(* IEC 61131-3 sources: Eaton-PLC-CSV-MQTT/CSV-MQTT/scripts/FunctionBlocks, 2 files *)

(* ---- FB_CSVReader.st ---- *)
// This function block reads CSV files row by row for PLC processing
// Uses state machine approach for efficient file handling
FUNCTION_BLOCK FB_CSVReader
VAR_INPUT
    xEnable   : BOOL;   // TRUE = start/continue reading, FALSE = stop and reset
    sFilePath : STRING; // File path to the CSV file (e.g., '/usr/data.csv')
END_VAR
VAR_OUTPUT
    RowOut    : ST_CSVRow; // Output: One parsed row with 13 columns of data
    xNewRow   : BOOL;      // Pulse TRUE when a new row is ready
    xBusy     : BOOL;      // TRUE while processing
    xError    : BOOL;      // TRUE if error occurred
    eError    : DWORD;     // Error code from file operations
    xDone     : BOOL;      // TRUE when finished reading entire file
END_VAR
VAR
    // State machine control
    eState : (IDLE, OPEN_FILE, READ_FILE, PARSE_LINES, CLOSE_FILE, ERROR) := IDLE;

    // File operation variables
    hFile      : DWORD := 16#FFFFFFFF; // File handle (using DWORD instead of RTS_IEC_HANDLE)
    sBuffer    : STRING(4096);   // Buffer for file content
    udiReadSize : UDINT;         // Actual bytes read
    diResult   : DINT;           // Function return values

    // Parsing variables
    iLineStart : INT := 1;       // Current position in buffer
    iLineEnd   : INT;            // End of current line
    sCurrentLine : STRING(512);  // Current line being processed
    iLineCount : INT := 0;       // Total lines processed
    bHeaderSkipped : BOOL := FALSE; // Track header skip

    // Control flags
    xEnableOld : BOOL := FALSE;  // Edge detection
END_VAR

// Reset on falling edge of xEnable
IF NOT xEnable AND xEnableOld THEN
    eState := IDLE;
    xBusy := FALSE;
    xError := FALSE;
    xDone := FALSE;
    xNewRow := FALSE;
    iLineStart := 1;
    iLineCount := 0;
    bHeaderSkipped := FALSE;
    IF hFile <> 16#FFFFFFFF THEN
        diResult := SysFileClose(hFile := hFile);
        hFile := 16#FFFFFFFF;
    END_IF;
END_IF;
xEnableOld := xEnable;

// State machine processing
xNewRow := FALSE; // Clear pulse output

CASE eState OF

    IDLE:
        IF xEnable THEN
            eState := OPEN_FILE;
            xBusy := TRUE;
            xError := FALSE;
            xDone := FALSE;
            sBuffer := '';
            iLineStart := 1;
        END_IF;

    OPEN_FILE:
        // Open file using SysFile function (not FB)
        hFile := SysFileOpen(szFile := sFilePath, am := 16#0001, pResult := ADR(diResult));
        IF hFile <> 16#FFFFFFFF THEN
            eState := READ_FILE;
        ELSE
            eError := DINT_TO_DWORD(diResult);
            xError := TRUE;
            eState := ERROR;
        END_IF;

    READ_FILE:
        // Read entire file content into buffer
        udiReadSize := SysFileRead(hFile := hFile, pbyBuffer := ADR(sBuffer),
                                    ulSize := SIZEOF(sBuffer)-1, pResult := ADR(diResult));
        IF diResult = 0 THEN
            eState := PARSE_LINES;
        ELSE
            eError := DINT_TO_DWORD(diResult);
            xError := TRUE;
            eState := CLOSE_FILE;
        END_IF;

    PARSE_LINES:
        // Extract next line from buffer
        IF F_GetNextLine(sBuffer := sBuffer, iStartPos := iLineStart,
                        sLine => sCurrentLine, iEndPos => iLineEnd) THEN
            iLineStart := iLineEnd + 1;
            iLineCount := iLineCount + 1;

            // Skip header row
            IF NOT bHeaderSkipped THEN
                bHeaderSkipped := TRUE;
            ELSE
                // Parse CSV line into structure
                RowOut := F_ParseCSVLine(sCurrentLine);
                xNewRow := TRUE; // Signal new row available
            END_IF;
        ELSE
            // No more lines - finished
            eState := CLOSE_FILE;
        END_IF;

    CLOSE_FILE:
        IF hFile <> 16#FFFFFFFF THEN
            diResult := SysFileClose(hFile := hFile);
            hFile := 16#FFFFFFFF;
        END_IF;
        xDone := TRUE;
        xBusy := FALSE;
        eState := IDLE;

    ERROR:
        xBusy := FALSE;
        IF hFile <> 16#FFFFFFFF THEN
            diResult := SysFileClose(hFile := hFile);
            hFile := 16#FFFFFFFF;
        END_IF;
        eState := IDLE;

END_CASE;

END_FUNCTION_BLOCK

(* ---- FB_MQTTPublisher.st ---- *)
// MQTT Publisher using Stefan Dreyer MQTT library
// Builds JSON from CSV row data and publishes it to the configured broker
FUNCTION_BLOCK FB_MQTTPublisher
VAR_INPUT
    xEnable       : BOOL;        // Enable MQTT connection
    xUseLaptop    : BOOL;        // TRUE = laptop connection, FALSE = router/LAN
    RowIn         : ST_CSVRow;   // CSV row data to publish
    xTrigger      : BOOL;        // Trigger to publish current row
    sBrokerLaptop : STRING(255) := 'broker.hivemq.com'; // Cloud broker for laptop mode
    sBrokerLAN    : STRING(255) := 'broker.hivemq.com'; // Cloud broker for LAN mode
    uiPort        : UINT := 1883; // MQTT port (1883 = no TLS)
    sTopic        : STRING(255) := 'UE/139ukr';      // MQTT topic
END_VAR
VAR_OUTPUT
    xConnected    : BOOL;        // TRUE when connected to broker
    xPublished    : BOOL;        // Pulse TRUE when message published
    xError        : BOOL;        // TRUE if error occurred
    sStatus       : STRING(128); // Status/error message
END_VAR
VAR
    // MQTT client structure and handler instances
    mqttInOut     : SD_MQTT.MQTT_IN_OUT;   // Shared MQTT data structure
    fbMQTTClient  : SD_MQTT.MqttClient;    // Main MQTT client FB
    fbMQTTPublish : SD_MQTT.MqttPublish;   // Publish helper FB

    // Connection / publish state machine
    eState        : (IDLE, CONNECTING, READY, PUBLISHING, ERROR) := IDLE;
    ePrevState    : (IDLE, CONNECTING, READY, PUBLISHING, ERROR) := IDLE;

    // Payload buffers
    sJsonPayload  : STRING(2048);
    sActiveTopic  : STRING(255);
    sActiveHost   : STRING(255);
    sUrlBuffer    : STRING(512);
    sPortBuffer   : STRING(16);

    // Helpers
    trigPublish   : Standard.R_TRIG;
    trigSend      : Standard.R_TRIG;
    xSendPulseReq : BOOL;
    xLinkDone     : BOOL;
    xUseTLS       : BOOL;
    xErrorLatched : BOOL;

    // MQTT client error latches
    dwClientError : DWORD;
    byClientError : BYTE;

    // Default QoS (0 = at most once)
    eDefaultQoS   : SD_MQTT.QoS := 0;
END_VAR
VAR CONSTANT
    c_tClientTimeout : TIME := T#5S;
END_VAR

// Clear pulse outputs each call
xPublished := FALSE;
xSendPulseReq := FALSE;

// Link publish FB once to the shared MQTT data
IF NOT xLinkDone THEN
    fbMQTTPublish.SetMqttInOut(MQTT_IN_OUT := mqttInOut);
    xLinkDone := TRUE;
END_IF;

// Select active host and client ID based on connection mode
IF xUseLaptop THEN
    sActiveHost := sBrokerLaptop;
    mqttInOut.ClientID := 'EatonPLC_Laptop';
ELSE
    sActiveHost := sBrokerLAN;
    mqttInOut.ClientID := 'EatonPLC_LAN';
END_IF;

// Align dynamic allocation limits with payload buffer size
mqttInOut.COM_CONFIG.MaxPayloadSize := UDINT#2048;

// Build URL in form host:port for client FB
sPortBuffer := UINT_TO_STRING(uiPort);
sUrlBuffer := Standard.CONCAT(STR1 := sActiveHost, STR2 := ':');
sUrlBuffer := Standard.CONCAT(STR1 := sUrlBuffer, STR2 := sPortBuffer);

// Enable TLS automatically for the standard secure port
xUseTLS := uiPort = 8883;

// Drive Stefan Dreyer MQTT client every cycle
fbMQTTClient(
    MQTT_IN_OUT := mqttInOut,
    ENABLE := xEnable,
    URL := sUrlBuffer,
    TIMEOUT := c_tClientTimeout,
    TLS := xUseTLS,
    ERROR_C => dwClientError,
    ERROR_T => byClientError
);

// Rising edge detection for publish trigger
trigPublish(CLK := xTrigger);

// State machine controlling connection and publish flow
CASE eState OF
    IDLE:
        xConnected := FALSE;
        IF NOT xEnable THEN
            xErrorLatched := FALSE;
            sStatus := 'Idle';
        ELSE
            sStatus := 'Connecting...';
            eState := CONNECTING;
        END_IF;

    CONNECTING:
        xConnected := FALSE;
        sStatus := 'Connecting...';
        IF NOT xEnable THEN
            eState := IDLE;
        ELSIF mqttInOut.BROKER_CONNECTED THEN
            sStatus := 'Connected';
            eState := READY;
        ELSIF (dwClientError <> DWORD#0) OR (byClientError <> BYTE#0) THEN
            xErrorLatched := TRUE;
            sStatus := 'Connection error';
            eState := ERROR;
        END_IF;

    READY:
        xConnected := TRUE;
        sStatus := 'Connected';
        IF NOT xEnable THEN
            eState := IDLE;
        ELSIF NOT mqttInOut.BROKER_CONNECTED THEN
            sStatus := 'Reconnecting...';
            eState := CONNECTING;
        ELSE
            // Keep local copy of topic while idle
            sActiveTopic := sTopic;

            IF trigPublish.Q THEN
                IF fbMQTTPublish.sendActive THEN
                    sStatus := 'Publish busy';
                ELSIF NOT F_BuildJsonFromRow(row := RowIn, sJson := sJsonPayload) THEN
                    xErrorLatched := TRUE;
                    sStatus := 'JSON build failed';
                    eState := ERROR;
                ELSE
                    xSendPulseReq := TRUE;
                    sStatus := 'Publishing...';
                    eState := PUBLISHING;
                END_IF;
            END_IF;
        END_IF;

    PUBLISHING:
        xConnected := mqttInOut.BROKER_CONNECTED;
        sStatus := 'Publishing...';
        IF NOT xEnable THEN
            eState := IDLE;
        ELSIF NOT mqttInOut.BROKER_CONNECTED THEN
            xErrorLatched := TRUE;
            sStatus := 'Connection lost';
            eState := ERROR;
        ELSIF fbMQTTPublish.done THEN
            xPublished := TRUE;
            sStatus := 'Published';
            eState := READY;
        ELSIF fbMQTTPublish.SendTimeout THEN
            xErrorLatched := TRUE;
            sStatus := 'Publish timeout';
            eState := ERROR;
        END_IF;

    ERROR:
        xConnected := FALSE;
        IF NOT xEnable THEN
            xErrorLatched := FALSE;
            sStatus := 'Idle';
            eState := IDLE;
        ELSIF (dwClientError <> DWORD#0) OR (byClientError <> BYTE#0) THEN
            sStatus := 'Client error';
        ELSE
            sStatus := 'Retrying...';
            eState := CONNECTING;
        END_IF;
END_CASE;

// Positive edge on publish send input
trigSend(CLK := xSendPulseReq);

// Execute publish FB (string payload mode)
fbMQTTPublish(
    Topic := ADR(sActiveTopic),
    PayloadString := ADR(sJsonPayload),
    PublishAsString := TRUE,
    Payload := 0,
    PayloadLength := 0,
    QoSIn := eDefaultQoS,
    MRetain := FALSE,
    send := trigSend.Q
);

// Clear latched error once stable connection restored
IF (ePrevState <> eState) AND (eState = READY) THEN
    xErrorLatched := FALSE;
END_IF;
ePrevState := eState;

// Final outputs
xConnected := xEnable AND mqttInOut.BROKER_CONNECTED;
xError := xErrorLatched OR (xEnable AND ((dwClientError <> DWORD#0) OR (byClientError <> BYTE#0)));

IF NOT xEnable THEN
    sStatus := 'Disabled';
END_IF;

END_FUNCTION_BLOCK
